// TIA Portal V17 export
// export: Created 2025-07-17T00:36:38.4776718Z, ExportSetting WithDefaults, DisplayName Totally Integrated Automation Portal, DisplayVersion V17, DisplayName TIA Portal Openness, DisplayVersion V17, DisplayName TIA Portal Version Control Interface, DisplayVersion V17, DisplayName STEP 7 Professional, DisplayVersion V17, DisplayName STEP 7 Safety, DisplayVersion V17, DisplayName WinCC Advanced / Unified PC, DisplayVersion V17
FUNCTION "pump_flow_set_and_read" : Void   // FC2, LAD
{ S7_Optimized_Access := 'TRUE' }
VERSION : 0.1
// stored: AutoNumber true, IsIECCheckEnabled false, SetENOAutomatically false, UDAEnableTagReadback false
   VAR_TEMP
      flow_read_temp1 : Real;
      flow_read_temp2 : Real;
      flow_read_temp3 : Real;
   END_VAR
BEGIN

REGION Network 1
   // 1号泵流量控制
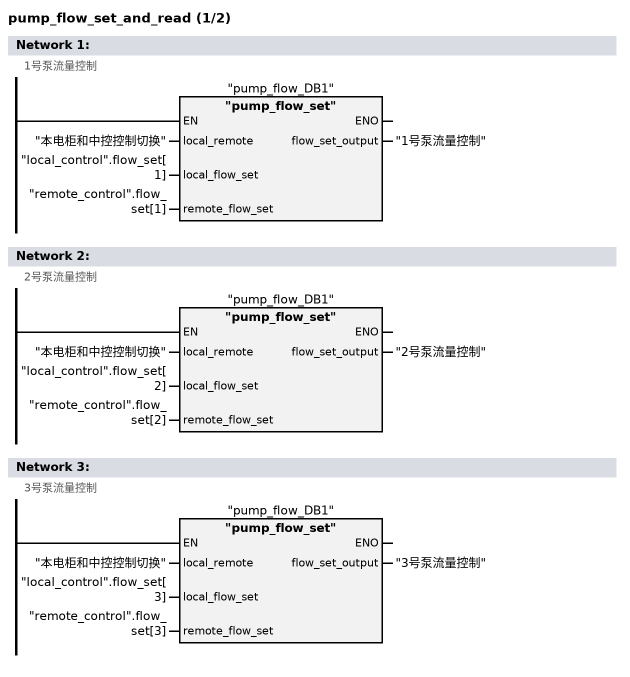
   RUNG wire#powerrail
      "pump_flow_DB1"(local_remote := "本电柜和中控控制切换", local_flow_set := "local_control".flow_set[1], remote_flow_set := "remote_control".flow_set[1], flow_set_output => "1号泵流量控制")
   END_RUNG
   // the same network as SCL:
   "pump_flow_DB1"(local_remote := "本电柜和中控控制切换",   // "pump_flow_set"
                   local_flow_set := "local_control".flow_set[1],
                   remote_flow_set := "remote_control".flow_set[1],
                   flow_set_output => "1号泵流量控制");
END_REGION

REGION Network 2
   // 2号泵流量控制
   RUNG wire#powerrail
      "pump_flow_DB1"(local_remote := "本电柜和中控控制切换", local_flow_set := "local_control".flow_set[2], remote_flow_set := "remote_control".flow_set[2], flow_set_output => "2号泵流量控制")
   END_RUNG
   // the same network as SCL:
   "pump_flow_DB1"(local_remote := "本电柜和中控控制切换",   // "pump_flow_set"
                   local_flow_set := "local_control".flow_set[2],
                   remote_flow_set := "remote_control".flow_set[2],
                   flow_set_output => "2号泵流量控制");
END_REGION

REGION Network 3
   // 3号泵流量控制
   RUNG wire#powerrail
      "pump_flow_DB1"(local_remote := "本电柜和中控控制切换", local_flow_set := "local_control".flow_set[3], remote_flow_set := "remote_control".flow_set[3], flow_set_output => "3号泵流量控制")
   END_RUNG
   // the same network as SCL:
   "pump_flow_DB1"(local_remote := "本电柜和中控控制切换",   // "pump_flow_set"
                   local_flow_set := "local_control".flow_set[3],
                   remote_flow_set := "remote_control".flow_set[3],
                   flow_set_output => "3号泵流量控制");
END_REGION

REGION Network 4
   // 读取计量泵反馈流量
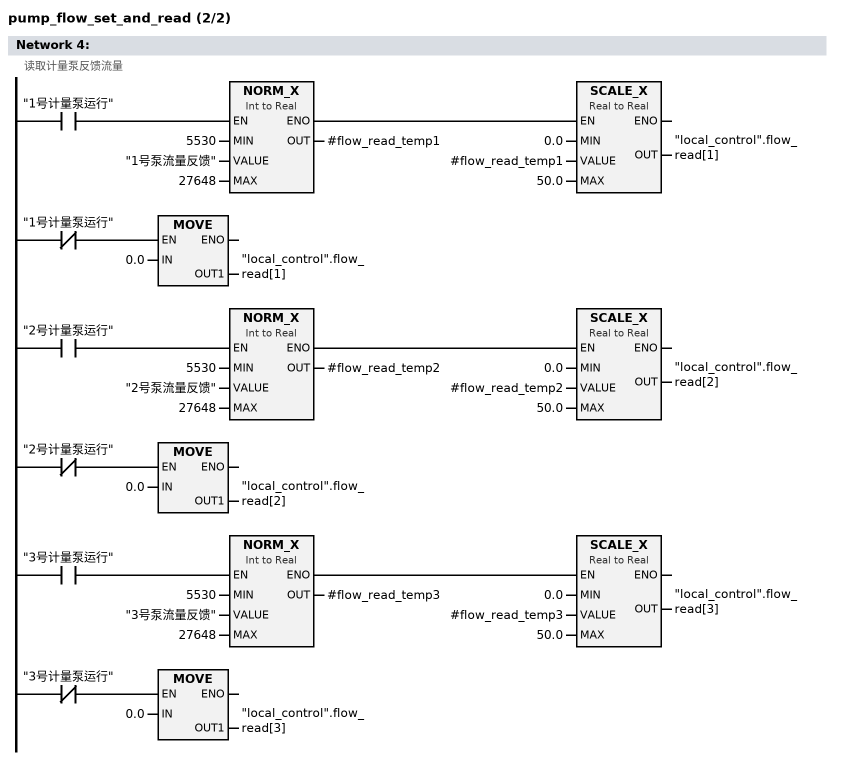
   RUNG wire#powerrail
      Contact( "1号计量泵运行" )
      { S7_Templates := "[SrcType := Int, DestType := Real]" } Normalize(min := 5530, value := "1号泵流量反馈", max := 27648, out => #flow_read_temp1)
      { S7_Templates := "[SrcType := Real, DestType := Real]" } Scale(min := 0.0, value := #flow_read_temp1, max := 50.0, out => "local_control".flow_read[1])
   END_RUNG
   RUNG wire#powerrail
      I_Contact( "1号计量泵运行" )
      Move(in := 0.0, out1 => "local_control".flow_read[1])
   END_RUNG
   RUNG wire#powerrail
      Contact( "2号计量泵运行" )
      { S7_Templates := "[SrcType := Int, DestType := Real]" } Normalize(min := 5530, value := "2号泵流量反馈", max := 27648, out => #flow_read_temp2)
      { S7_Templates := "[SrcType := Real, DestType := Real]" } Scale(min := 0.0, value := #flow_read_temp2, max := 50.0, out => "local_control".flow_read[2])
   END_RUNG
   RUNG wire#powerrail
      I_Contact( "2号计量泵运行" )
      Move(in := 0.0, out1 => "local_control".flow_read[2])
   END_RUNG
   RUNG wire#powerrail
      Contact( "3号计量泵运行" )
      { S7_Templates := "[SrcType := Int, DestType := Real]" } Normalize(min := 5530, value := "3号泵流量反馈", max := 27648, out => #flow_read_temp3)
      { S7_Templates := "[SrcType := Real, DestType := Real]" } Scale(min := 0.0, value := #flow_read_temp3, max := 50.0, out => "local_control".flow_read[3])
   END_RUNG
   RUNG wire#powerrail
      I_Contact( "3号计量泵运行" )
      Move(in := 0.0, out1 => "local_control".flow_read[3])
   END_RUNG
   // the same network as SCL:
   IF "1号计量泵运行" THEN
       #flow_read_temp1 := NORM_X(MIN := 5530, VALUE := "1号泵流量反馈", MAX := 27648);
       "local_control".flow_read[1] := SCALE_X(MIN := 0.0, VALUE := #flow_read_temp1, MAX := 50.0);
   END_IF;
   IF NOT "1号计量泵运行" THEN "local_control".flow_read[1] := 0.0; END_IF;
   IF "2号计量泵运行" THEN
       #flow_read_temp2 := NORM_X(MIN := 5530, VALUE := "2号泵流量反馈", MAX := 27648);
       "local_control".flow_read[2] := SCALE_X(MIN := 0.0, VALUE := #flow_read_temp2, MAX := 50.0);
   END_IF;
   IF NOT "2号计量泵运行" THEN "local_control".flow_read[2] := 0.0; END_IF;
   IF "3号计量泵运行" THEN
       #flow_read_temp3 := NORM_X(MIN := 5530, VALUE := "3号泵流量反馈", MAX := 27648);
       "local_control".flow_read[3] := SCALE_X(MIN := 0.0, VALUE := #flow_read_temp3, MAX := 50.0);
   END_IF;
   IF NOT "3号计量泵运行" THEN "local_control".flow_read[3] := 0.0; END_IF;
END_REGION
END_FUNCTION
